PROGRAM P_Demo_FIX16Sub
VAR
    fp8A     : T_FIX16;
    fp8B     : T_FIX16;
    fp8Diff  : T_FIX16;
    lrResult : LREAL;
    bSub     : BOOL;
END_VAR

// ============================================================
// Tc2_Utilities.FIX16Sub 演示程序（FUNCTION，单周期触发）
// ============================================================
// 场景：读两个传感器之差用于偏差控制。
// 价值：替代手写对齐 + INT 减法。
// 验证步骤：
//   1. 把本 PROGRAM 加到 PlcTask 调用列表
//   2. 编译 + 登录
//   3. 在线把 b... 触发位置 TRUE 一个周期
//   4. 观察输出变量是否符合期望
// ============================================================

fp8A := LREAL_TO_FIX16(0.5,  8);
fp8B := LREAL_TO_FIX16(0.75, 8);
IF bSub THEN
    fp8Diff  := FIX16Sub(fp8A, fp8B);
    lrResult := FIX16_TO_LREAL(fp8Diff);   // 应为 -0.25
    bSub := FALSE;
END_IF;

END_PROGRAM

(* stored: Version 1.1.0.1, ProductVersion 3.1.4024.5
   POU P_Demo_FIX16Sub: Id {4493dfbe-2b72-513f-ab3e-8743c66264c6}, SpecialFunc None *)
